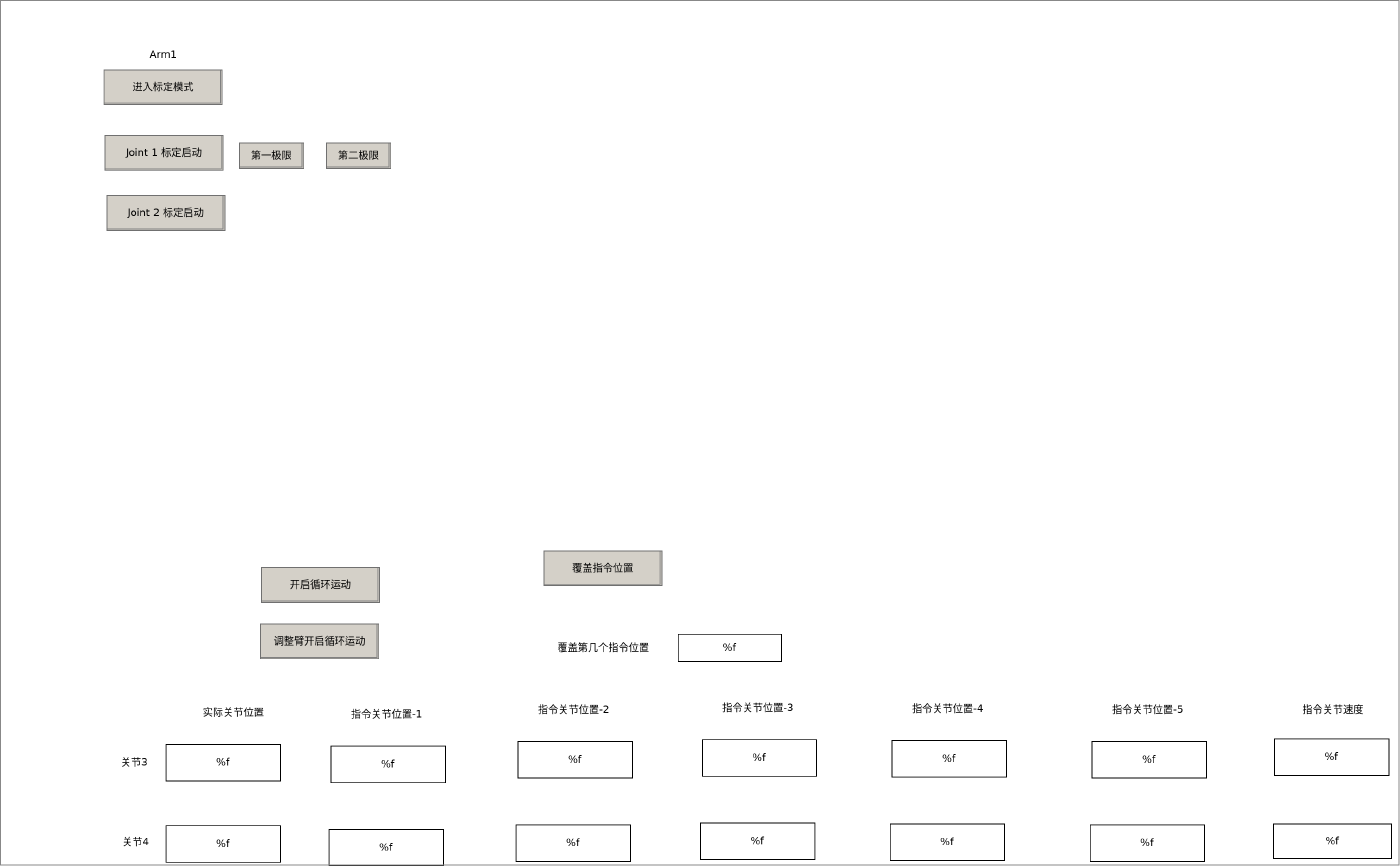
VISUALIZATION arm4Cail  // 1512x936
    Button (112,75 128x38), "进入标定模式", colour toggle: g_cycleTest.m_enterCycleTestMode[1]
        toggle g_cycleTest.m_enterCycleTestMode[1]
    Button (282,613 128x38), "开启循环运动", colour toggle: g_cycleTest.m_startMotion[1]
        toggle g_cycleTest.m_startMotion[1]
    Label (345,758 145x28), "指令关节位置-1"
    Label (177,755 150x30), "实际关节位置"
    Label (115,810 60x28), "关节3"
    Label (119,896 55x28), "关节4"
    Rectangle (179,804 124x40), "%f", text variable: g_cycleTest.m_actJntPosSetup[1][3]
    Rectangle (179,892 124x40), "%f", text variable: g_cycleTest.m_actJntPosSetup[1][4]
    Rectangle (357,806 124x40), "%f", text variable: g_cycleTest.m_targetJntPosSetup[1,1][3]
        OnMouseClick: write the text variable via Default
    Rectangle (355,896 124x40), "%f", text variable: g_cycleTest.m_targetJntPosSetup[1,1][4]
        OnMouseClick: write the text variable via Default
    Label (547,753 145x28), "指令关节位置-2"
    Rectangle (559,801 124x40), "%f", text variable: g_cycleTest.m_targetJntPosSetup[1,2][3]
        OnMouseClick: write the text variable via Default
    Rectangle (557,891 124x40), "%f", text variable: g_cycleTest.m_targetJntPosSetup[1,2][4]
        OnMouseClick: write the text variable via Default
    Label (746,751 145x28), "指令关节位置-3"
    Rectangle (758,799 124x40), "%f", text variable: g_cycleTest.m_targetJntPosSetup[1,3][3]
        OnMouseClick: write the text variable via Default
    Rectangle (756,889 124x40), "%f", text variable: g_cycleTest.m_targetJntPosSetup[1,3][4]
        OnMouseClick: write the text variable via Default
    Label (951,752 145x28), "指令关节位置-4"
    Rectangle (963,800 124x40), "%f", text variable: g_cycleTest.m_targetJntPosSetup[1,4][3]
        OnMouseClick: write the text variable via Default
    Rectangle (961,890 124x40), "%f", text variable: g_cycleTest.m_targetJntPosSetup[1,4][4]
        OnMouseClick: write the text variable via Default
    Label (1167,753 145x28), "指令关节位置-5"
    Rectangle (1179,801 124x40), "%f", text variable: g_cycleTest.m_targetJntPosSetup[1,5][3]
        OnMouseClick: write the text variable via Default
    Rectangle (1177,891 124x40), "%f", text variable: g_cycleTest.m_targetJntPosSetup[1,5][4]
        OnMouseClick: write the text variable via Default
    Button (113,146 128x38), "Joint 1 标定启动", colour toggle: g_cycleTest.m_enterCycleTestModeSetup[1]
        toggle g_cycleTest.m_enterCycleTestModeSetup[1]
    Button (281,674 128x38), "调整臂开启循环运动", colour toggle: g_cycleTest.m_startMotionSetup[1]
        toggle g_cycleTest.m_startMotionSetup[1]
    Button (587,595 128x38), "覆盖指令位置", colour toggle: g_cycleTest.m_coverCmdPos[1]
        tap g_cycleTest.m_coverCmdPos[1]
    Rectangle (732,685 112x30), "%f", text variable: g_cycleTest.m_pntIdForCoverCmd[1]
        OnMouseClick: write the text variable via Default
    Label (579,686 145x28), "覆盖第几个指令位置"
    Label (1367,753 145x28), "指令关节速度"
    Rectangle (1376,798 124x40), "%f", text variable: g_cycleTest.m_targetJntVelSetup[1][3]
        OnMouseClick: write the text variable via Default
    Rectangle (1375,890 128x38), "%f", text variable: g_cycleTest.m_targetJntVelSetup[1][4]
        OnMouseClick: write the text variable via Default
    Label (131,47 91x24), "Arm1"
    Button (115,211 128x38), "Joint 2 标定启动", colour toggle: g_cycleTest.m_enterCycleTestModeSetup[1]
        toggle g_cycleTest.m_enterCycleTestModeSetup[1]
    Button (258,154 70x28), "第一极限", colour toggle: g_cycleTest.m_enterCycleTestModeSetup[1]
        toggle g_cycleTest.m_enterCycleTestModeSetup[1]
    Button (352,154 70x28), "第二极限", colour toggle: g_cycleTest.m_enterCycleTestModeSetup[1]
        toggle g_cycleTest.m_enterCycleTestModeSetup[1]
END_VISUALIZATION

(* stored: Version 1.1.0.1, ProductVersion 3.1.4024.11
   Visu arm4Cail: Id {6869464a-52a9-47ff-a1c6-4f2cfc1cb5ec} *)
